SUBAPPLICATION GreenWhiteBackground_Schneidwerk (* Subapplication Type *)
  (* Standard: 61499-2 *)
  (* Version 1.0, 2023-02-11, franz *)
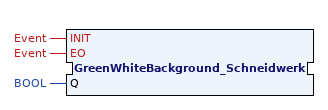
  EVENT_INPUT
    INIT;
    EO;
  END_EVENT
  VAR_INPUT
    Q : BOOL;
  END_VAR
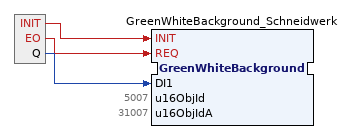
  SUBAPPS
    GreenWhiteBackground_Schneidwerk : GreenWhiteBackground(u16ObjId := 5007, u16ObjIdA := 31007);
  END_SUBAPPS
  EVENT_CONNECTIONS
    INIT TO GreenWhiteBackground_Schneidwerk.INIT;
    EO TO GreenWhiteBackground_Schneidwerk.REQ;
  END_CONNECTIONS
  DATA_CONNECTIONS
    Q TO GreenWhiteBackground_Schneidwerk.DI1;
  END_CONNECTIONS
END_SUBAPPLICATION
